INTERFACE I_CamCurveComp EXTENDS I_SequenceTest

END_INTERFACE

(* stored: Version 1.1.0.1, ProductVersion 3.1.4026.19
   Itf I_CamCurveComp: Id {9a82bb89-62ce-4f1e-8de6-fc8e5e003e1b} *)
